
// ===== library: MasterCopy "FB_SP-CLP" =====

// folder: 08_Comunicação/SP-CLP

FUNCTION_BLOCK "FB_SP-CLP"   // FB10, SCL
{ S7_Optimized_Access := 'FALSE' }
VERSION : 0.1
   VAR_INPUT
      Auto : Bool;
      Run : Bool;
      Fault : Bool;
      Safety : Bool;
      "Counter" : Bool;
      Signal_5 : Bool;
      Signal_6 : Bool;
      Signal_7 : Bool;
      Signal_8 : Bool;
      Signal_9 : Bool;
      Signal_10 : Bool;
      Signal_11 : Bool;
      Signal_12 : Bool;
      Signal_13 : Bool;
      Signal_14 : Bool;
      Signal_15 : Bool;
      DInt_1 : DInt;
      DInt_2 : DInt;
      DInt_3 : DInt;
   END_VAR
   VAR_OUTPUT
      "Type" : Array[0..4] of Char;
      Count : DInt;
   END_VAR
   VAR
      CountProd : IEC_UDCOUNTER;
   END_VAR
   VAR_TEMP
      PV : Int;
      HabCounter : Bool;
   END_VAR
   // "Type"[0] := 'S';
   // "Type"[1] := 'P';
   // "Type"[2] := 'C';
   // "Type"[3] := 'L';
   // "Type"[4] := 'P';
BEGIN
   #CountProd.R := "FirstScan";

   IF #Run THEN
       "#CountProd".CTU(CU := #Counter,
                        PV := #PV,
                        R := "FirstScan",
                        CV => #Count);
   END_IF;
END_FUNCTION_BLOCK